// TIA Portal project "Projekt 2, grundprogram" (V16)

(* hardware
DEVICE "S71500/ET200MP station_1"  S7-1500 station
   slot 0: "Rail_0"  6ES7 590-1***0-0AA0
   slot 1: "PLC_2 Sortering"  CPU 1516-3 PN/DP  6ES7 516-3AN01-0AB0  V2.0
      slot 3: "CPU display_1"  6ES7591-1BA00-0AA0
      slot 32768: "PROFINET interface_1"  X1
         slot 32769: "Port_1"  X1 P1
         slot 32770: "Port_2"  X1 P2
      slot 33024: "PROFINET interface_2"  X2
         slot 33025: "Port_1"  X2 P1
      slot 33280: "DP interface_1"  X3
   slot 2: "DI 32x24VDC HF_1"  DI 32x24VDC HF  6ES7 521-1BL00-0AB0  V2.0
   slot 3: "DQ 32x24VDC/0.5A HF_1"  DQ 32x24VDC/0.5A HF  6ES7 522-1BL01-0AB0  V1.0
   slot 4: "AI 8xU/I/RTD/TC ST_1"  AI 8xU/I/RTD/TC ST  6ES7 531-7KF00-0AB0  V2.0
   slot 5: "AQ 4xU/I ST_1"  AQ 4xU/I ST  6ES7 532-5HD00-0AB0  V2.0
DEVICE "S71500/ET200MP station_2"  S7-1500 station
   slot 0: "Rail_0"  6ES7 590-1***0-0AA0
   slot 1: "PLC_1 Inspektion"  CPU 1516-3 PN/DP  6ES7 516-3AN01-0AB0  V2.0
      slot 3: "CPU display_1"  6ES7591-1BA00-0AA0
      slot 32768: "PROFINET interface_1"  X1
         slot 32769: "Port_1"  X1 P1
         slot 32770: "Port_2"  X1 P2
      slot 33024: "PROFINET interface_2"  X2
         slot 33025: "Port_1"  X2 P1
      slot 33280: "DP interface_1"  X3
   slot 2: "DI 32x24VDC HF_1"  DI 32x24VDC HF  6ES7 521-1BL00-0AB0  V2.0
   slot 3: "DQ 32x24VDC/0.5A HF_1"  DQ 32x24VDC/0.5A HF  6ES7 522-1BL01-0AB0  V1.0
   slot 4: "AI 8xU/I/RTD/TC ST_1"  AI 8xU/I/RTD/TC ST  6ES7 531-7KF00-0AB0  V2.0
   slot 5: "AQ 4xU/I ST_1"  AQ 4xU/I ST  6ES7 532-5HD00-0AB0  V2.0
*)

// ===== PLC "PLC_2 Sortering"  CPU 1516-3 PN/DP =====

VAR_GLOBAL   // PLC tag table "Default tag table"
   "System_Byte" AT %MB1 : Byte;
   "FirstScan" AT %M1.0 : Bool;
   "DiagStatusUpdate" AT %M1.1 : Bool;
   "AlwaysTRUE" AT %M1.2 : Bool;
   "AlwaysFALSE" AT %M1.3 : Bool;
   "Clock_Byte" AT %MB0 : Byte;
   "Clock_10Hz" AT %M0.0 : Bool;
   "Clock_5Hz" AT %M0.1 : Bool;
   "Clock_2.5Hz" AT %M0.2 : Bool;
   "Clock_2Hz" AT %M0.3 : Bool;
   "Clock_1.25Hz" AT %M0.4 : Bool;
   "Clock_1Hz" AT %M0.5 : Bool;
   "Clock_0.625Hz" AT %M0.6 : Bool;
   "Clock_0.5Hz" AT %M0.7 : Bool;
   "Tag_1" AT %IB0 : Byte;
   "Tag_2" AT %QB0 : Byte;
   "Tag_3" AT %IB1 : Byte;
   "Tag_4" AT %QB1 : Byte;
   "Tag_5" AT %IB2 : Byte;
   "Tag_6" AT %IB3 : Byte;
END_VAR

VAR_GLOBAL   // PLC tag table "Fysiske IO"
   "Anden fotocelle" AT %I0.0 : Bool;   // NO
   "Første fotocelle" AT %I0.1 : Bool;   // NO
   "Fotocelle over adskiller" AT %I0.2 : Bool;   // NC OBS. Desuden ind på XMA3(C)
   "Induktiv aftaster på akuator til fjernelse af emne" AT %I0.3 : Bool;   // Signal ON ved upåvirket aktuator
   "Fotocelle på sidebånd" AT %I0.4 : Bool;   // NC
   "Fotocelle efter udskydning til sidebånd" AT %I0.5 : Bool;   // NC
   "Hovedtransportbånd" AT %Q0.0 : Bool;
   "Sidetransportbånd" AT %Q0.1 : Bool;
   "Aktuator til frigivelse på hovedbånd" AT %Q0.2 : Bool;   // Er ude i upåvirket tilstand
   "Aktuator til udskydning til sidebånd" AT %Q0.3 : Bool;   // Lige gennemgang i upåvirket tilstand
END_VAR

ORGANIZATION_BLOCK "Main"   // OB1, FBD, ProgramCycle
TITLE = "Main Program Sweep (Cycle)"
{ S7_Optimized_Access := 'TRUE' }
VERSION : 0.1
   VAR_INPUT
      Initial_Call : Bool;   // Initial call of this OB
      Remanence : Bool;   // =True, if remanent data are available
   END_VAR
BEGIN
END_ORGANIZATION_BLOCK

// ===== PLC "PLC_1 Inspektion"  CPU 1516-3 PN/DP =====

VAR_GLOBAL   // PLC tag table "Default tag table"
   "System_Byte" AT %MB1 : Byte;
   "FirstScan" AT %M1.0 : Bool;
   "DiagStatusUpdate" AT %M1.1 : Bool;
   "AlwaysTRUE" AT %M1.2 : Bool;
   "AlwaysFALSE" AT %M1.3 : Bool;
   "Clock_Byte" AT %MB0 : Byte;
   "Clock_10Hz" AT %M0.0 : Bool;
   "Clock_5Hz" AT %M0.1 : Bool;
   "Clock_2.5Hz" AT %M0.2 : Bool;
   "Clock_2Hz" AT %M0.3 : Bool;
   "Clock_1.25Hz" AT %M0.4 : Bool;
   "Clock_1Hz" AT %M0.5 : Bool;
   "Clock_0.625Hz" AT %M0.6 : Bool;
   "Clock_0.5Hz" AT %M0.7 : Bool;
   "Tag_1" AT %IB0 : Byte;
   "Tag_2" AT %QB0 : Byte;
   "Tag_3" AT %IB1 : Byte;
   "Tag_4" AT %QB1 : Byte;
   "Tag_5" AT %IB2 : Byte;
   "Tag_6" AT %IB3 : Byte;
END_VAR

VAR_GLOBAL   // PLC tag table "Fysiske IO"
   "Første fotocelle" AT %I0.0 : Bool;
   "Fotocelle ved adskiller" AT %I0.1 : Bool;   // NO
   "Sidste fotocelle" AT %I0.2 : Bool;   // NC
   "Cylinder ved føder er upåvirket" AT %I0.4 : Bool;   // Bruges ikke
   "Cylinder ved føder er påvirket" AT %I0.5 : Bool;   // Bruges ikke
   "Lager indeholde emne" AT %I0.6 : Bool;   // Bruges ikke
   "Transportbånd, frem" AT %Q0.0 : Bool;
   "Transportbånd, tilbage" AT %Q0.1 : Bool;
   "Adskiller" AT %Q0.2 : Bool;
   "Cylinder på føder" AT %Q0.4 : Bool;   // Bruges ikke
END_VAR

ORGANIZATION_BLOCK "Main"   // OB1, FBD, ProgramCycle
TITLE = "Main Program Sweep (Cycle)"
{ S7_Optimized_Access := 'TRUE' }
VERSION : 0.1
   VAR_INPUT
      Initial_Call : Bool;   // Initial call of this OB
      Remanence : Bool;   // =True, if remanent data are available
   END_VAR
BEGIN
END_ORGANIZATION_BLOCK